Yaskawa INFORM job: R1_ISOPOUNCE.JBI

/JOB
//NAME R1_ISOPOUNCE
//POS
///NPOS 0,0,0,0,0,0
//INST
///DATE 2021/09/30 10:12
///ATTR SC,RW
///GROUP1 RB1
///LVARS 0,0,0,0,0,0,0,0
NOP
'%%%%%%%%%%%%%%%%%%%%%%%%%%%%%%%%
' R1 ISO Pounce Position
'%%%%%%%%%%%%%%%%%%%%%%%%%%%%%%%%
'
*TOP
'***********INITIALIZE***********
' Set Clear of Module Bits
CALL JOB:R1_CLEARMODULE ARGF235
' Report Position
CALL JOB:R1_REPORTPOS ARGF3
'********************************
'
'********PRE-STATUS_CHECK********
'********************************
'
'***********PRIME_MOVE***********
'********************************
MOVJ P[106] VJ=25.00
'
'*******POST-STATUS_CHECK********
'********************************
'
'****USER_DEFINED_PARAMETERS*****
'********************************
'
'********DATA_VALIDATION*********
'********************************
'
'*************SETUP**************
'********************************
'
'*************ACTION*************
'********************************
'
'*********HOUSE_KEEPING**********
SET B004 1
'********************************
*OUT
END
